% RSLogix 500 project VA116HF7_OPRAVOVANY_4_2017_02_12.rss, saved by version 8.40.00.08 %
PROJECT "VA116"    % processor: SLC 500, 1747-L532; 601760_CO2 %

PROGRAM FILES
  LAD 2 "601760_CO2"  92 rungs
  LAD 3   24 rungs
  LAD 4   108 rungs
  LAD 5   16 rungs
  LAD 6   98 rungs
  LAD 7   26 rungs
  LAD 8   13 rungs
  LAD 9   15 rungs
  LAD 10   50 rungs
  LAD 11   95 rungs
  LAD 12   18 rungs
  LAD 13   34 rungs
  LAD 14   6 rungs
  LAD 15   28 rungs
  LAD 16   84 rungs
  LAD 17   22 rungs
  LAD 18   23 rungs
  LAD 19   37 rungs
  LAD 20   5 rungs
  LAD 21   19 rungs
  LAD 22   29 rungs
  LAD 23   17 rungs
  LAD 24   32 rungs
  LAD 25   8 rungs
  LAD 26   57 rungs
  LAD 27   4 rungs
  LAD 28   3 rungs
  LAD 29   4 rungs
  LAD 30   12 rungs
  LAD 31   12 rungs
  LAD 32   22 rungs
  LAD 33   10 rungs
  LAD 34   16 rungs
  LAD 35   14 rungs

DATA FILES
  O0 OUTPUT  4 elements
  I1 INPUT  8 elements
  S2 STATUS  83 elements
  B3 BINARY  1 elements
  T4 TIMER  61 elements
  C5 COUNTER  6 elements
  R6 CONTROL  1 elements
  N7 INTEGER  110 elements
  N10   256 elements
  N11   256 elements

LADDER 2 "601760_CO2"
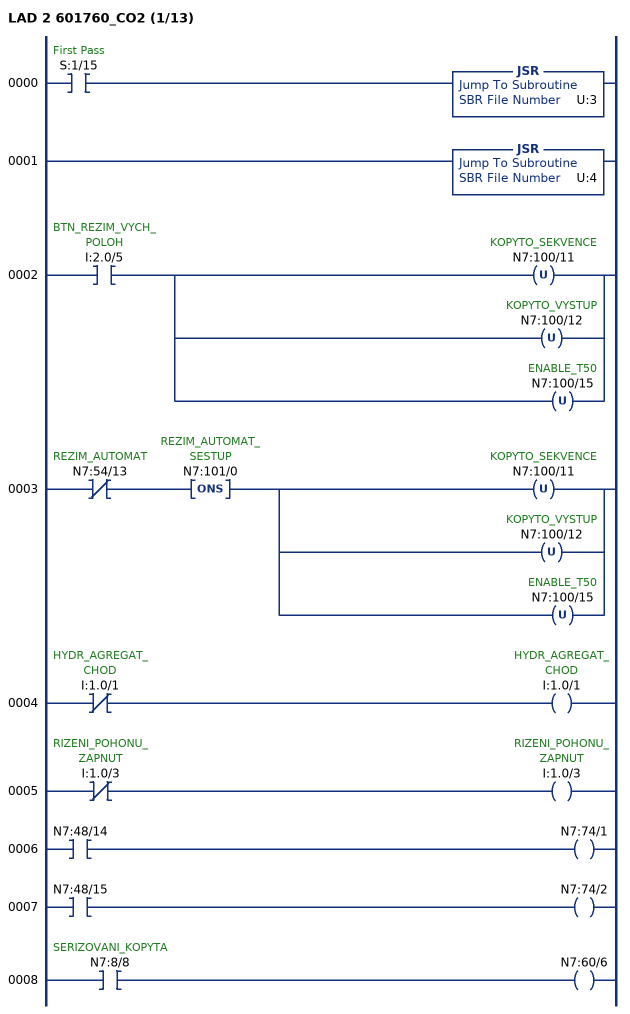
% Rung: 0 %
SOR XIC S:1/15 JSR U:3 EOR
%   S:1/15  "First Pass" %
% Rung: 1 %
SOR JSR U:4 EOR
% Rung: 2 %
SOR XIC I:2.0/5 BST OTU N7:100/11 NXB OTU N7:100/12 NXB OTU N7:100/15 BND EOR
%   I:2.0/5  BTN_REZIM_VYCH_POLOH %
%   N7:100/11  KOPYTO_SEKVENCE %
%   N7:100/12  KOPYTO_VYSTUP %
%   N7:100/15  ENABLE_T50 %
% Rung: 3 %
SOR XIO N7:54/13 OSR N7:101/0 BST OTU N7:100/11 NXB OTU N7:100/12 NXB OTU N7:100/15 BND EOR
%   N7:54/13  REZIM_AUTOMAT %
%   N7:101/0  REZIM_AUTOMAT_SESTUP %
%   N7:100/11  KOPYTO_SEKVENCE %
%   N7:100/12  KOPYTO_VYSTUP %
%   N7:100/15  ENABLE_T50 %
% Rung: 4 %
SOR XIO I:1.0/1 OTE I:1.0/1 EOR
%   I:1.0/1  HYDR_AGREGAT_CHOD %
% Rung: 5 %
SOR XIO I:1.0/3 OTE I:1.0/3 EOR
%   I:1.0/3  RIZENI_POHONU_ZAPNUT %
% Rung: 6 %
SOR XIC N7:48/14 OTE N7:74/1 EOR
% Rung: 7 %
SOR XIC N7:48/15 OTE N7:74/2 EOR
% Rung: 8 %
SOR XIC N7:8/8 OTE N7:60/6 EOR
%   N7:8/8  SERIZOVANI_KOPYTA %

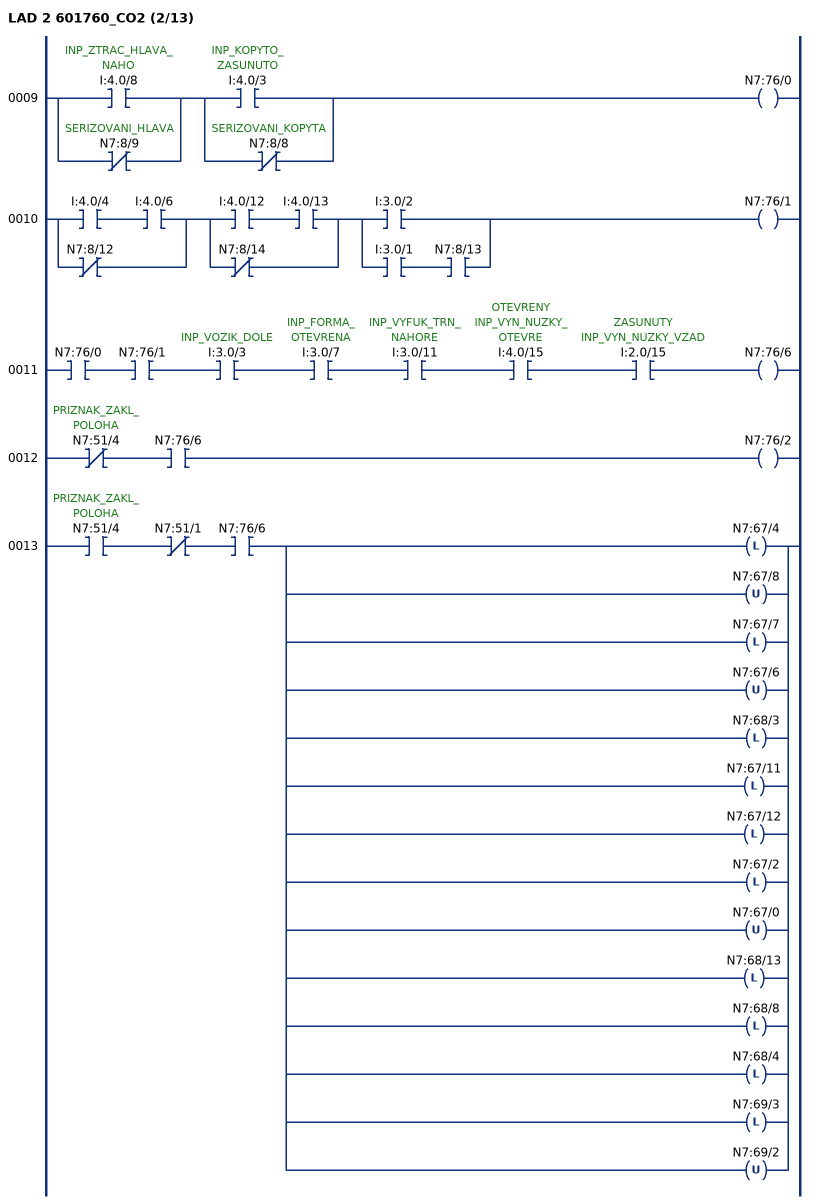
% Rung: 9 %
SOR BST XIC I:4.0/8 NXB XIO N7:8/9 BND BST XIC I:4.0/3 NXB XIO N7:8/8 BND OTE N7:76/0 EOR
%   I:4.0/8  INP_ZTRAC_HLAVA_NAHO %
%   N7:8/9  SERIZOVANI_HLAVA %
%   I:4.0/3  INP_KOPYTO_ZASUNUTO %
%   N7:8/8  SERIZOVANI_KOPYTA %
% Rung: 10 %
SOR BST XIC I:4.0/4 XIC I:4.0/6 NXB XIO N7:8/12 BND BST XIC I:4.0/12 XIC I:4.0/13 NXB XIO N7:8/14 BND BST XIC I:3.0/2 NXB XIC I:3.0/1 XIC N7:8/13 BND OTE N7:76/1 EOR
% Rung: 11 %
SOR XIC N7:76/0 XIC N7:76/1 XIC I:3.0/3 XIC I:3.0/7 XIC I:3.0/11 XIC I:4.0/15 XIC I:2.0/15 OTE N7:76/6 EOR
%   I:3.0/3  INP_VOZIK_DOLE %
%   I:3.0/7  INP_FORMA_OTEVRENA %
%   I:3.0/11  INP_VYFUK_TRN_NAHORE %
%   I:4.0/15  INP_VYN_NUZKY_OTEVRE  "OTEVRENY" %
%   I:2.0/15  INP_VYN_NUZKY_VZAD  "ZASUNUTY" %
% Rung: 12 %
SOR XIO N7:51/4 XIC N7:76/6 OTE N7:76/2 EOR
%   N7:51/4  PRIZNAK_ZAKL_POLOHA %
% Rung: 13 %
SOR XIC N7:51/4 XIO N7:51/1 XIC N7:76/6 BST OTL N7:67/4 NXB OTU N7:67/8 NXB BST OTL N7:67/7 NXB OTU N7:67/6 BND NXB OTL N7:68/3 NXB OTL N7:67/11 NXB OTL N7:67/12 NXB OTL N7:67/2 NXB OTU N7:67/0 NXB OTL N7:68/13 NXB OTL N7:68/8 NXB BST OTL N7:68/4 NXB BST OTL N7:69/3 NXB OTU N7:69/2 BND BND BND EOR
%   N7:51/4  PRIZNAK_ZAKL_POLOHA %

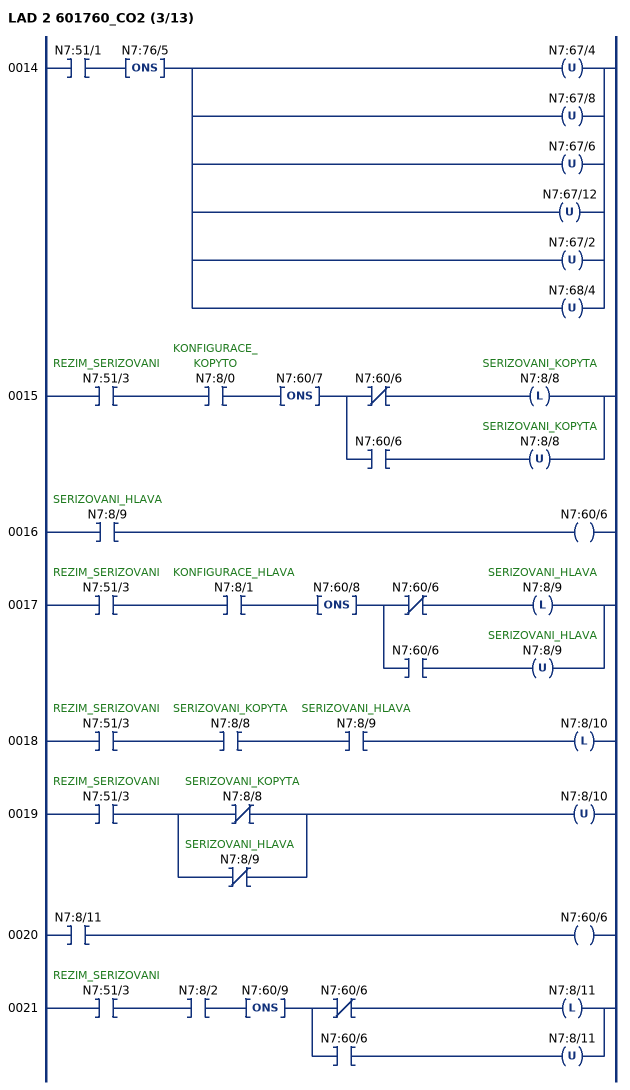
% Rung: 14 %
SOR XIC N7:51/1 OSR N7:76/5 BST OTU N7:67/4 NXB OTU N7:67/8 NXB OTU N7:67/6 NXB OTU N7:67/12 NXB OTU N7:67/2 NXB OTU N7:68/4 BND EOR
% Rung: 15 %
SOR XIC N7:51/3 XIC N7:8/0 OSR N7:60/7 BST XIO N7:60/6 OTL N7:8/8 NXB XIC N7:60/6 OTU N7:8/8 BND EOR
%   N7:51/3  REZIM_SERIZOVANI %
%   N7:8/0  KONFIGURACE_KOPYTO %
%   N7:8/8  SERIZOVANI_KOPYTA %
% Rung: 16 %
SOR XIC N7:8/9 OTE N7:60/6 EOR
%   N7:8/9  SERIZOVANI_HLAVA %
% Rung: 17 %
SOR XIC N7:51/3 XIC N7:8/1 OSR N7:60/8 BST XIO N7:60/6 OTL N7:8/9 NXB XIC N7:60/6 OTU N7:8/9 BND EOR
%   N7:51/3  REZIM_SERIZOVANI %
%   N7:8/1  KONFIGURACE_HLAVA %
%   N7:8/9  SERIZOVANI_HLAVA %
% Rung: 18 %
SOR XIC N7:51/3 XIC N7:8/8 XIC N7:8/9 OTL N7:8/10 EOR
%   N7:51/3  REZIM_SERIZOVANI %
%   N7:8/8  SERIZOVANI_KOPYTA %
%   N7:8/9  SERIZOVANI_HLAVA %
% Rung: 19 %
SOR XIC N7:51/3 BST XIO N7:8/8 NXB XIO N7:8/9 BND OTU N7:8/10 EOR
%   N7:51/3  REZIM_SERIZOVANI %
%   N7:8/8  SERIZOVANI_KOPYTA %
%   N7:8/9  SERIZOVANI_HLAVA %
% Rung: 20 %
SOR XIC N7:8/11 OTE N7:60/6 EOR
% Rung: 21 %
SOR XIC N7:51/3 XIC N7:8/2 OSR N7:60/9 BST XIO N7:60/6 OTL N7:8/11 NXB XIC N7:60/6 OTU N7:8/11 BND EOR
%   N7:51/3  REZIM_SERIZOVANI %

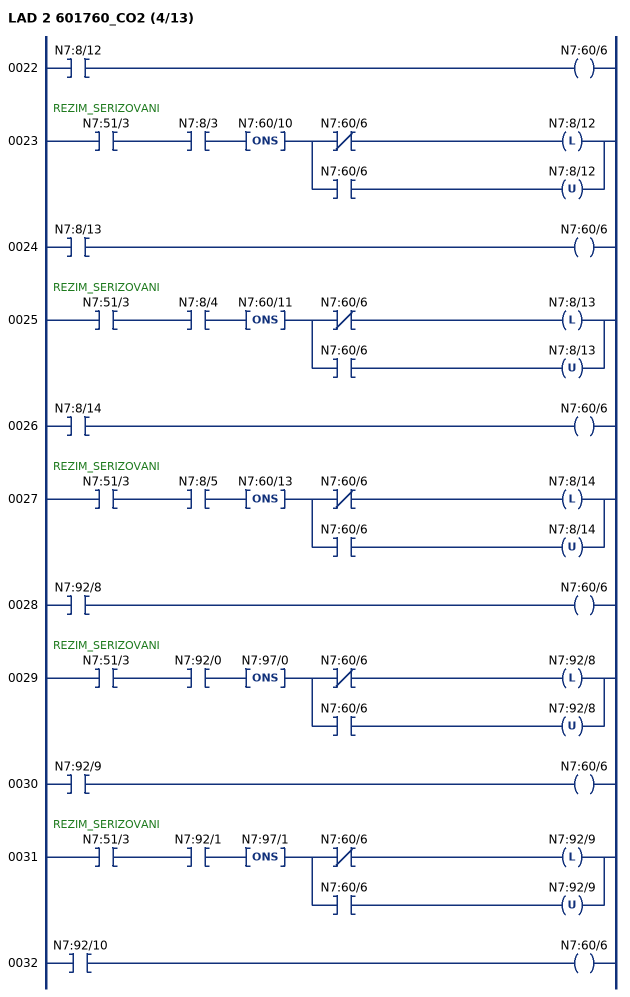
% Rung: 22 %
SOR XIC N7:8/12 OTE N7:60/6 EOR
% Rung: 23 %
SOR XIC N7:51/3 XIC N7:8/3 OSR N7:60/10 BST XIO N7:60/6 OTL N7:8/12 NXB XIC N7:60/6 OTU N7:8/12 BND EOR
%   N7:51/3  REZIM_SERIZOVANI %
% Rung: 24 %
SOR XIC N7:8/13 OTE N7:60/6 EOR
% Rung: 25 %
SOR XIC N7:51/3 XIC N7:8/4 OSR N7:60/11 BST XIO N7:60/6 OTL N7:8/13 NXB XIC N7:60/6 OTU N7:8/13 BND EOR
%   N7:51/3  REZIM_SERIZOVANI %
% Rung: 26 %
SOR XIC N7:8/14 OTE N7:60/6 EOR
% Rung: 27 %
SOR XIC N7:51/3 XIC N7:8/5 OSR N7:60/13 BST XIO N7:60/6 OTL N7:8/14 NXB XIC N7:60/6 OTU N7:8/14 BND EOR
%   N7:51/3  REZIM_SERIZOVANI %
% Rung: 28 %
SOR XIC N7:92/8 OTE N7:60/6 EOR
% Rung: 29 %
SOR XIC N7:51/3 XIC N7:92/0 OSR N7:97/0 BST XIO N7:60/6 OTL N7:92/8 NXB XIC N7:60/6 OTU N7:92/8 BND EOR
%   N7:51/3  REZIM_SERIZOVANI %
% Rung: 30 %
SOR XIC N7:92/9 OTE N7:60/6 EOR
% Rung: 31 %
SOR XIC N7:51/3 XIC N7:92/1 OSR N7:97/1 BST XIO N7:60/6 OTL N7:92/9 NXB XIC N7:60/6 OTU N7:92/9 BND EOR
%   N7:51/3  REZIM_SERIZOVANI %
% Rung: 32 %
SOR XIC N7:92/10 OTE N7:60/6 EOR

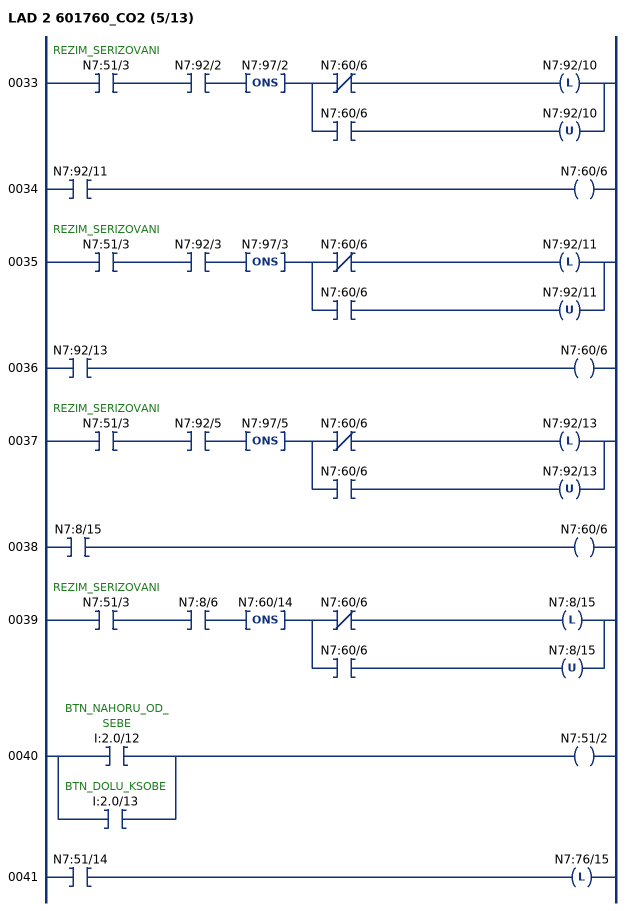
% Rung: 33 %
SOR XIC N7:51/3 XIC N7:92/2 OSR N7:97/2 BST XIO N7:60/6 OTL N7:92/10 NXB XIC N7:60/6 OTU N7:92/10 BND EOR
%   N7:51/3  REZIM_SERIZOVANI %
% Rung: 34 %
SOR XIC N7:92/11 OTE N7:60/6 EOR
% Rung: 35 %
SOR XIC N7:51/3 XIC N7:92/3 OSR N7:97/3 BST XIO N7:60/6 OTL N7:92/11 NXB XIC N7:60/6 OTU N7:92/11 BND EOR
%   N7:51/3  REZIM_SERIZOVANI %
% Rung: 36 %
SOR XIC N7:92/13 OTE N7:60/6 EOR
% Rung: 37 %
SOR XIC N7:51/3 XIC N7:92/5 OSR N7:97/5 BST XIO N7:60/6 OTL N7:92/13 NXB XIC N7:60/6 OTU N7:92/13 BND EOR
%   N7:51/3  REZIM_SERIZOVANI %
% Rung: 38 %
SOR XIC N7:8/15 OTE N7:60/6 EOR
% Rung: 39 %
SOR XIC N7:51/3 XIC N7:8/6 OSR N7:60/14 BST XIO N7:60/6 OTL N7:8/15 NXB XIC N7:60/6 OTU N7:8/15 BND EOR
%   N7:51/3  REZIM_SERIZOVANI %
% Rung: 40 %
SOR BST XIC I:2.0/12 NXB XIC I:2.0/13 BND OTE N7:51/2 EOR
%   I:2.0/12  BTN_NAHORU_OD_SEBE %
%   I:2.0/13  BTN_DOLU_KSOBE %
% Rung: 41 %
SOR XIC N7:51/14 OTL N7:76/15 EOR

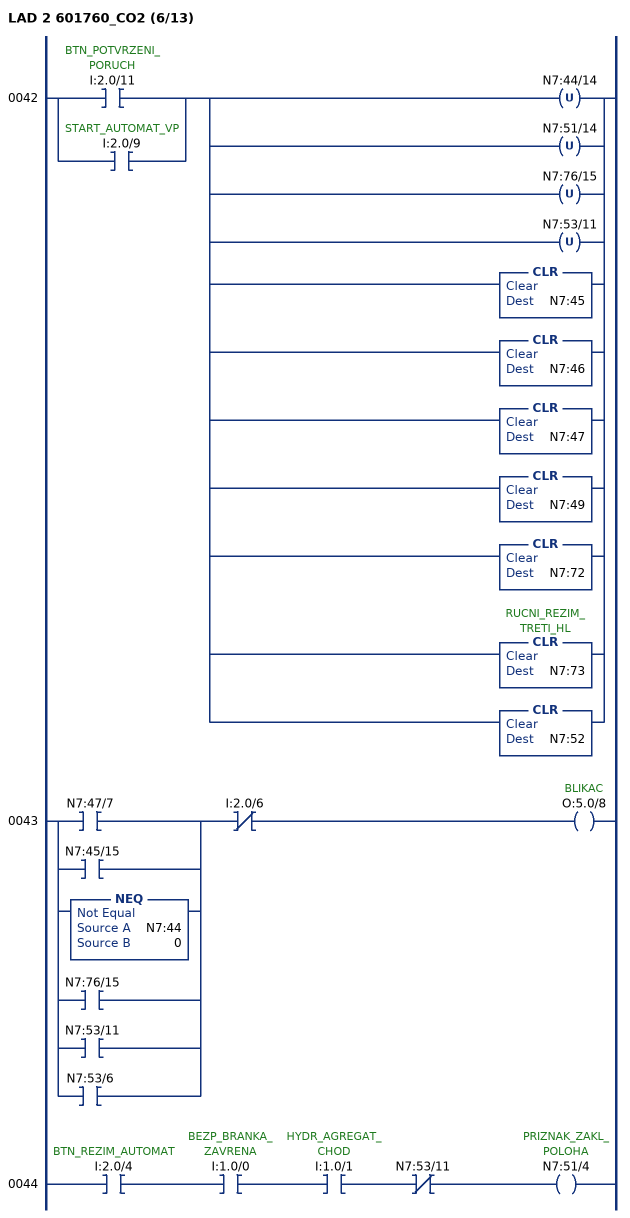
% Rung: 42 %
SOR BST XIC I:2.0/11 NXB XIC I:2.0/9 BND BST OTU N7:44/14 NXB OTU N7:51/14 NXB OTU N7:76/15 NXB OTU N7:53/11 NXB CLR N7:45 NXB CLR N7:46 NXB CLR N7:47 NXB CLR N7:49 NXB CLR N7:72 NXB CLR N7:73 NXB CLR N7:52 BND EOR
%   I:2.0/11  BTN_POTVRZENI_PORUCH %
%   I:2.0/9  START_AUTOMAT_VP %
%   N7:73  RUCNI_REZIM_TRETI_HL %
% Rung: 43 %
SOR BST XIC N7:47/7 NXB XIC N7:45/15 NXB NEQ N7:44 0 NXB XIC N7:76/15 NXB XIC N7:53/11 NXB XIC N7:53/6 BND XIO I:2.0/6 OTE O:5.0/8 EOR
%   O:5.0/8  BLIKAC %
% Rung: 44 %
SOR XIC I:2.0/4 XIC I:1.0/0 XIC I:1.0/1 XIO N7:53/11 OTE N7:51/4 EOR
%   I:2.0/4  BTN_REZIM_AUTOMAT %
%   I:1.0/0  BEZP_BRANKA_ZAVRENA %
%   I:1.0/1  HYDR_AGREGAT_CHOD %
%   N7:51/4  PRIZNAK_ZAKL_POLOHA %

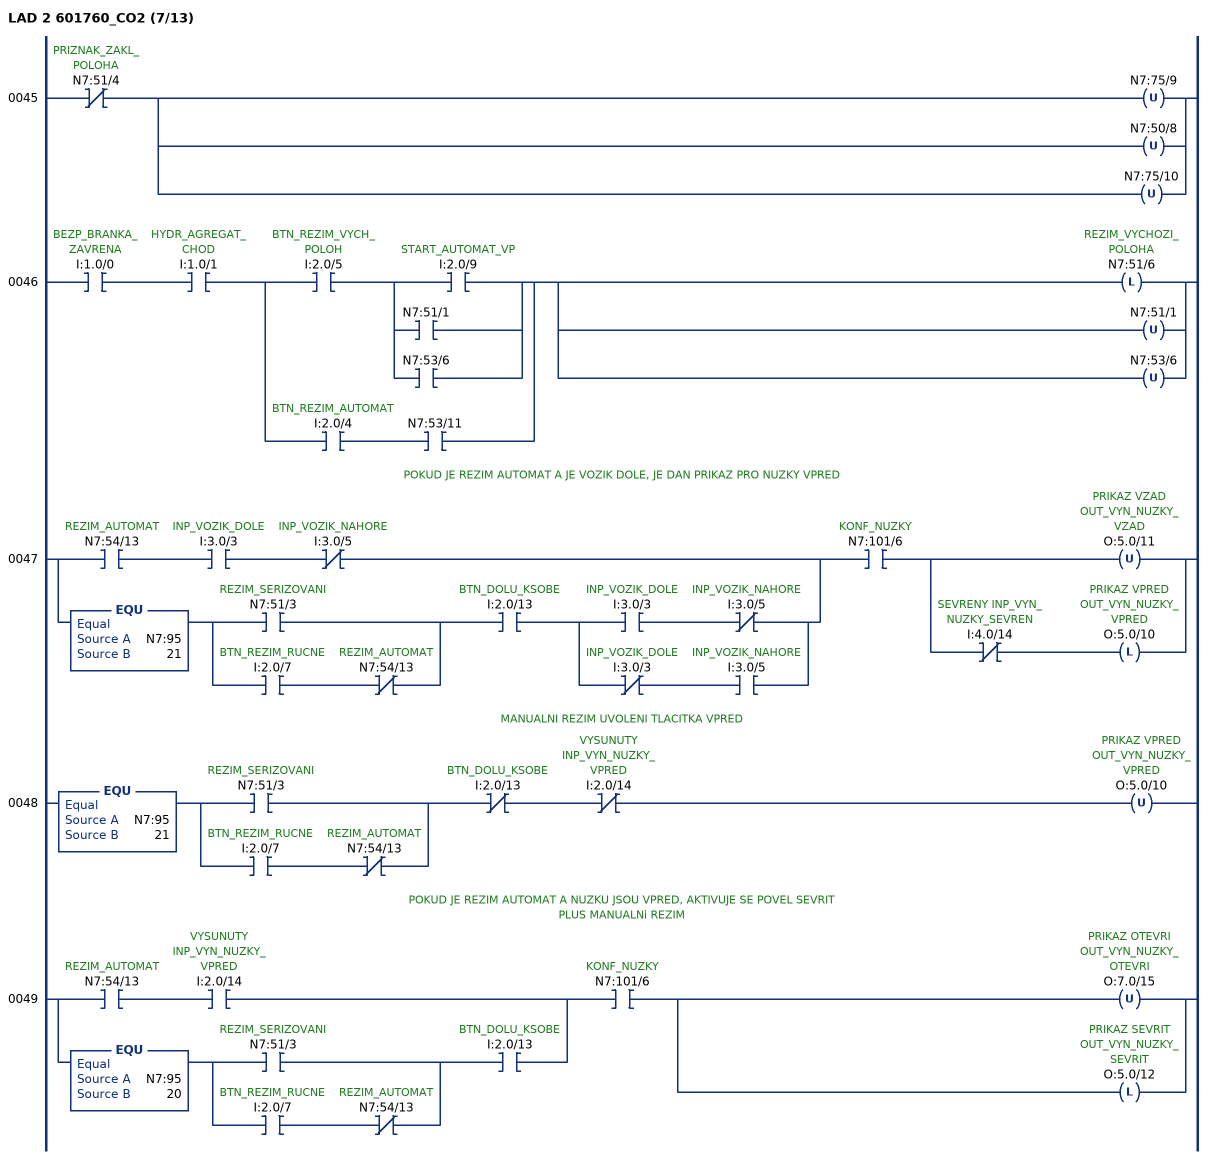
% Rung: 45 %
SOR XIO N7:51/4 BST OTU N7:75/9 NXB OTU N7:50/8 NXB OTU N7:75/10 BND EOR
%   N7:51/4  PRIZNAK_ZAKL_POLOHA %
% Rung: 46 %
SOR XIC I:1.0/0 XIC I:1.0/1 BST XIC I:2.0/5 BST XIC I:2.0/9 NXB XIC N7:51/1 NXB XIC N7:53/6 BND NXB XIC I:2.0/4 XIC N7:53/11 BND BST OTL N7:51/6 NXB OTU N7:51/1 NXB OTU N7:53/6 BND EOR
%   I:1.0/0  BEZP_BRANKA_ZAVRENA %
%   I:1.0/1  HYDR_AGREGAT_CHOD %
%   I:2.0/5  BTN_REZIM_VYCH_POLOH %
%   I:2.0/9  START_AUTOMAT_VP %
%   I:2.0/4  BTN_REZIM_AUTOMAT %
%   N7:51/6  REZIM_VYCHOZI_POLOHA %
% Rung: 47 %
% POKUD JE REZIM AUTOMAT A JE VOZIK DOLE, JE DAN PRIKAZ PRO NUZKY VPRED %
SOR BST XIC N7:54/13 XIC I:3.0/3 XIO I:3.0/5 NXB EQU N7:95 21 BST XIC N7:51/3 NXB XIC I:2.0/7 XIO N7:54/13 BND XIC I:2.0/13 BST XIC I:3.0/3 XIO I:3.0/5 NXB XIO I:3.0/3 XIC I:3.0/5 BND BND XIC N7:101/6 BST OTU O:5.0/11 NXB XIO I:4.0/14 OTL O:5.0/10 BND EOR
%   N7:54/13  REZIM_AUTOMAT %
%   I:3.0/3  INP_VOZIK_DOLE %
%   I:3.0/5  INP_VOZIK_NAHORE %
%   N7:51/3  REZIM_SERIZOVANI %
%   I:2.0/7  BTN_REZIM_RUCNE %
%   I:2.0/13  BTN_DOLU_KSOBE %
%   N7:101/6  KONF_NUZKY %
%   O:5.0/11  OUT_VYN_NUZKY_VZAD  "PRIKAZ VZAD" %
%   I:4.0/14  INP_VYN_NUZKY_SEVREN  "SEVRENY" %
%   O:5.0/10  OUT_VYN_NUZKY_VPRED  "PRIKAZ VPRED" %
% Rung: 48 %
% MANUALNI REZIM UVOLENI TLACITKA VPRED %
SOR EQU N7:95 21 BST XIC N7:51/3 NXB XIC I:2.0/7 XIO N7:54/13 BND XIO I:2.0/13 XIO I:2.0/14 OTU O:5.0/10 EOR
%   N7:51/3  REZIM_SERIZOVANI %
%   I:2.0/7  BTN_REZIM_RUCNE %
%   N7:54/13  REZIM_AUTOMAT %
%   I:2.0/13  BTN_DOLU_KSOBE %
%   I:2.0/14  INP_VYN_NUZKY_VPRED  "VYSUNUTY" %
%   O:5.0/10  OUT_VYN_NUZKY_VPRED  "PRIKAZ VPRED" %
% Rung: 49 %
% POKUD JE REZIM AUTOMAT A NUZKU JSOU VPRED, AKTIVUJE SE POVEL SEVRIT
% PLUS MANUALNi REZIM %
SOR BST XIC N7:54/13 XIC I:2.0/14 NXB EQU N7:95 20 BST XIC N7:51/3 NXB XIC I:2.0/7 XIO N7:54/13 BND XIC I:2.0/13 BND XIC N7:101/6 BST OTU O:7.0/15 NXB OTL O:5.0/12 BND EOR
%   N7:54/13  REZIM_AUTOMAT %
%   I:2.0/14  INP_VYN_NUZKY_VPRED  "VYSUNUTY" %
%   N7:51/3  REZIM_SERIZOVANI %
%   I:2.0/7  BTN_REZIM_RUCNE %
%   I:2.0/13  BTN_DOLU_KSOBE %
%   N7:101/6  KONF_NUZKY %
%   O:7.0/15  OUT_VYN_NUZKY_OTEVRI  "PRIKAZ OTEVRI" %
%   O:5.0/12  OUT_VYN_NUZKY_SEVRIT  "PRIKAZ SEVRIT" %

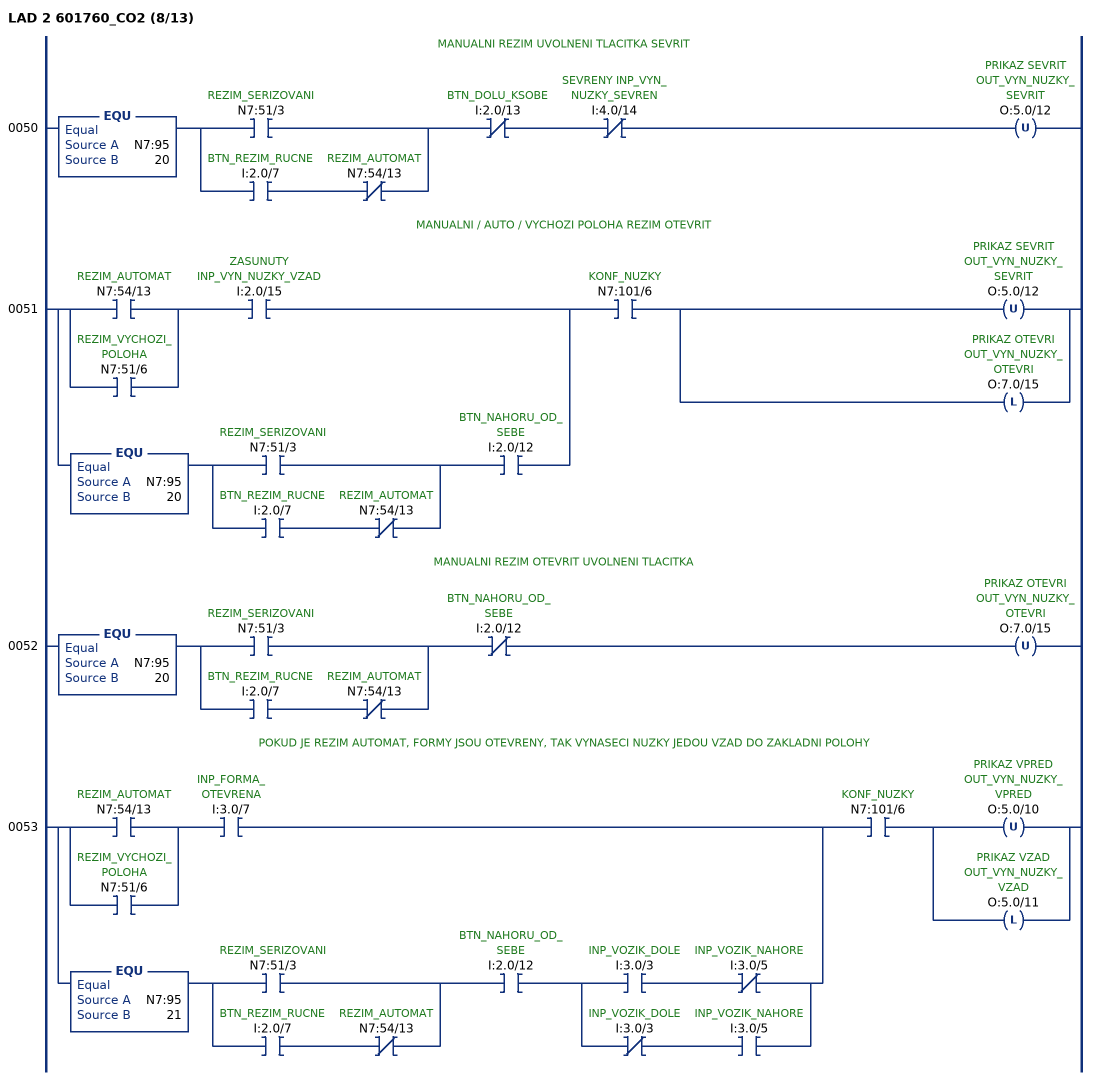
% Rung: 50 %
% MANUALNI REZIM UVOLNENI TLACITKA SEVRIT %
SOR EQU N7:95 20 BST XIC N7:51/3 NXB XIC I:2.0/7 XIO N7:54/13 BND XIO I:2.0/13 XIO I:4.0/14 OTU O:5.0/12 EOR
%   N7:51/3  REZIM_SERIZOVANI %
%   I:2.0/7  BTN_REZIM_RUCNE %
%   N7:54/13  REZIM_AUTOMAT %
%   I:2.0/13  BTN_DOLU_KSOBE %
%   I:4.0/14  INP_VYN_NUZKY_SEVREN  "SEVRENY" %
%   O:5.0/12  OUT_VYN_NUZKY_SEVRIT  "PRIKAZ SEVRIT" %
% Rung: 51 %
% MANUALNI / AUTO / VYCHOZI POLOHA REZIM OTEVRIT %
SOR BST BST XIC N7:54/13 NXB XIC N7:51/6 BND XIC I:2.0/15 NXB EQU N7:95 20 BST XIC N7:51/3 NXB XIC I:2.0/7 XIO N7:54/13 BND XIC I:2.0/12 BND XIC N7:101/6 BST OTU O:5.0/12 NXB OTL O:7.0/15 BND EOR
%   N7:54/13  REZIM_AUTOMAT %
%   N7:51/6  REZIM_VYCHOZI_POLOHA %
%   I:2.0/15  INP_VYN_NUZKY_VZAD  "ZASUNUTY" %
%   N7:51/3  REZIM_SERIZOVANI %
%   I:2.0/7  BTN_REZIM_RUCNE %
%   I:2.0/12  BTN_NAHORU_OD_SEBE %
%   N7:101/6  KONF_NUZKY %
%   O:5.0/12  OUT_VYN_NUZKY_SEVRIT  "PRIKAZ SEVRIT" %
%   O:7.0/15  OUT_VYN_NUZKY_OTEVRI  "PRIKAZ OTEVRI" %
% Rung: 52 %
% MANUALNI REZIM OTEVRIT UVOLNENI TLACITKA %
SOR EQU N7:95 20 BST XIC N7:51/3 NXB XIC I:2.0/7 XIO N7:54/13 BND XIO I:2.0/12 OTU O:7.0/15 EOR
%   N7:51/3  REZIM_SERIZOVANI %
%   I:2.0/7  BTN_REZIM_RUCNE %
%   N7:54/13  REZIM_AUTOMAT %
%   I:2.0/12  BTN_NAHORU_OD_SEBE %
%   O:7.0/15  OUT_VYN_NUZKY_OTEVRI  "PRIKAZ OTEVRI" %
% Rung: 53 %
% POKUD JE REZIM AUTOMAT, FORMY JSOU OTEVRENY, TAK VYNASECI NUZKY JEDOU VZAD DO ZAKLADNI POLOHY %
SOR BST BST XIC N7:54/13 NXB XIC N7:51/6 BND XIC I:3.0/7 NXB EQU N7:95 21 BST XIC N7:51/3 NXB XIC I:2.0/7 XIO N7:54/13 BND XIC I:2.0/12 BST XIC I:3.0/3 XIO I:3.0/5 NXB XIO I:3.0/3 XIC I:3.0/5 BND BND XIC N7:101/6 BST OTU O:5.0/10 NXB OTL O:5.0/11 BND EOR
%   N7:54/13  REZIM_AUTOMAT %
%   N7:51/6  REZIM_VYCHOZI_POLOHA %
%   I:3.0/7  INP_FORMA_OTEVRENA %
%   N7:51/3  REZIM_SERIZOVANI %
%   I:2.0/7  BTN_REZIM_RUCNE %
%   I:2.0/12  BTN_NAHORU_OD_SEBE %
%   I:3.0/3  INP_VOZIK_DOLE %
%   I:3.0/5  INP_VOZIK_NAHORE %
%   N7:101/6  KONF_NUZKY %
%   O:5.0/10  OUT_VYN_NUZKY_VPRED  "PRIKAZ VPRED" %
%   O:5.0/11  OUT_VYN_NUZKY_VZAD  "PRIKAZ VZAD" %

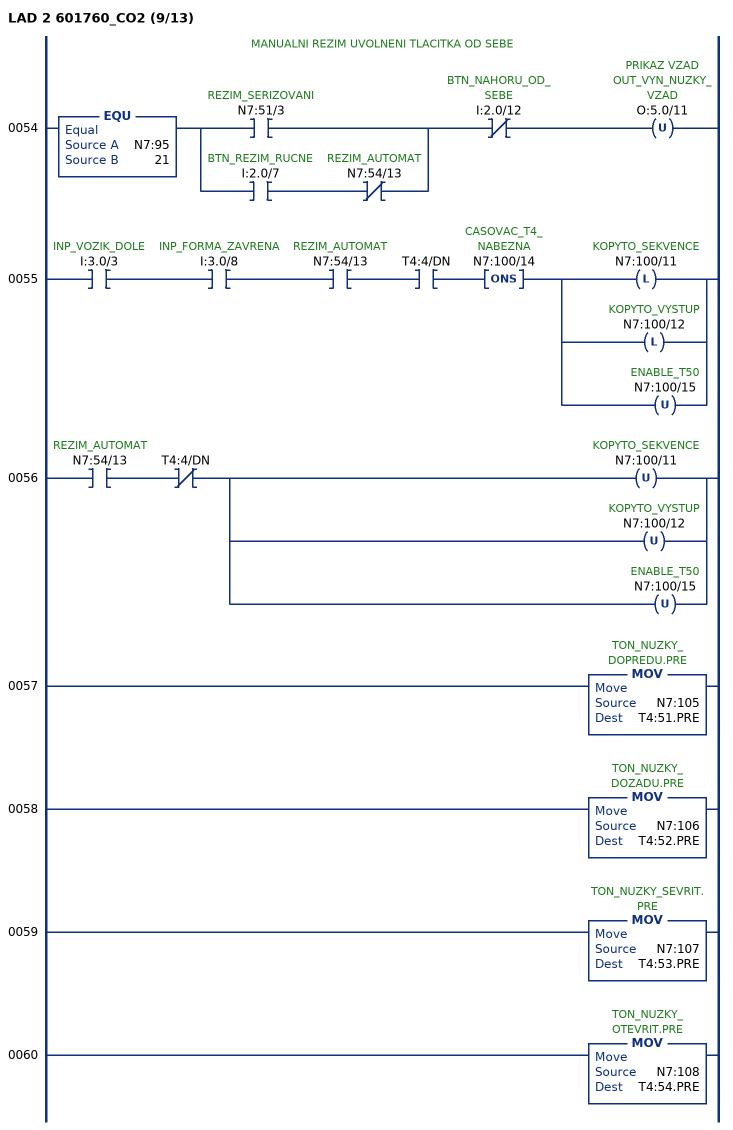
% Rung: 54 %
% MANUALNI REZIM UVOLNENI TLACITKA OD SEBE %
SOR EQU N7:95 21 BST XIC N7:51/3 NXB XIC I:2.0/7 XIO N7:54/13 BND XIO I:2.0/12 OTU O:5.0/11 EOR
%   N7:51/3  REZIM_SERIZOVANI %
%   I:2.0/7  BTN_REZIM_RUCNE %
%   N7:54/13  REZIM_AUTOMAT %
%   I:2.0/12  BTN_NAHORU_OD_SEBE %
%   O:5.0/11  OUT_VYN_NUZKY_VZAD  "PRIKAZ VZAD" %
% Rung: 55 %
SOR XIC I:3.0/3 XIC I:3.0/8 XIC N7:54/13 XIC T4:4/DN OSR N7:100/14 BST OTL N7:100/11 NXB OTL N7:100/12 NXB OTU N7:100/15 BND EOR
%   I:3.0/3  INP_VOZIK_DOLE %
%   I:3.0/8  INP_FORMA_ZAVRENA %
%   N7:54/13  REZIM_AUTOMAT %
%   N7:100/14  CASOVAC_T4_NABEZNA %
%   N7:100/11  KOPYTO_SEKVENCE %
%   N7:100/12  KOPYTO_VYSTUP %
%   N7:100/15  ENABLE_T50 %
% Rung: 56 %
SOR XIC N7:54/13 XIO T4:4/DN BST OTU N7:100/11 NXB OTU N7:100/12 NXB OTU N7:100/15 BND EOR
%   N7:54/13  REZIM_AUTOMAT %
%   N7:100/11  KOPYTO_SEKVENCE %
%   N7:100/12  KOPYTO_VYSTUP %
%   N7:100/15  ENABLE_T50 %
% Rung: 57 %
SOR MOV N7:105 T4:51.PRE EOR
%   N7:105  CASOVAC_T51_PRESET %
%   T4:51  TON_NUZKY_DOPREDU %
% Rung: 58 %
SOR MOV N7:106 T4:52.PRE EOR
%   N7:106  CASOVAC_T52_PRESET %
%   T4:52  TON_NUZKY_DOZADU %
% Rung: 59 %
SOR MOV N7:107 T4:53.PRE EOR
%   N7:107  CASOVAC_T53_PRESET %
%   T4:53  TON_NUZKY_SEVRIT %
% Rung: 60 %
SOR MOV N7:108 T4:54.PRE EOR
%   N7:108  CASOVAC_T54_PRESET %
%   T4:54  TON_NUZKY_OTEVRIT %

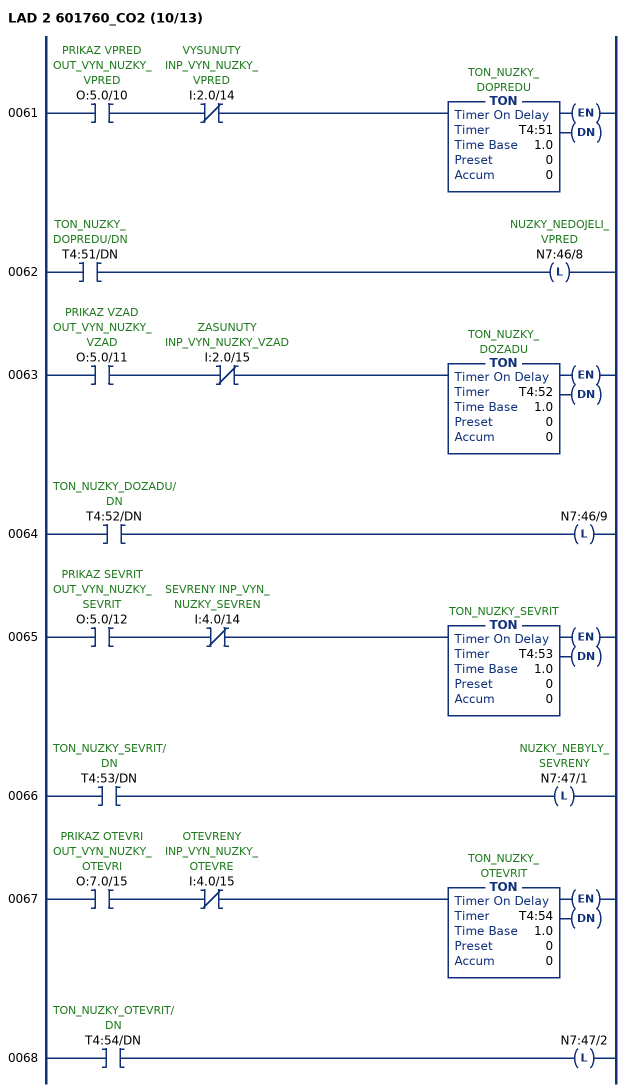
% Rung: 61 %
SOR XIC O:5.0/10 XIO I:2.0/14 TON T4:51 1.0 0 0 EOR
%   O:5.0/10  OUT_VYN_NUZKY_VPRED  "PRIKAZ VPRED" %
%   I:2.0/14  INP_VYN_NUZKY_VPRED  "VYSUNUTY" %
%   T4:51  TON_NUZKY_DOPREDU %
% Rung: 62 %
SOR XIC T4:51/DN OTL N7:46/8 EOR
%   T4:51  TON_NUZKY_DOPREDU %
%   N7:46/8  NUZKY_NEDOJELI_VPRED %
% Rung: 63 %
SOR XIC O:5.0/11 XIO I:2.0/15 TON T4:52 1.0 0 0 EOR
%   O:5.0/11  OUT_VYN_NUZKY_VZAD  "PRIKAZ VZAD" %
%   I:2.0/15  INP_VYN_NUZKY_VZAD  "ZASUNUTY" %
%   T4:52  TON_NUZKY_DOZADU %
% Rung: 64 %
SOR XIC T4:52/DN OTL N7:46/9 EOR
%   T4:52  TON_NUZKY_DOZADU %
% Rung: 65 %
SOR XIC O:5.0/12 XIO I:4.0/14 TON T4:53 1.0 0 0 EOR
%   O:5.0/12  OUT_VYN_NUZKY_SEVRIT  "PRIKAZ SEVRIT" %
%   I:4.0/14  INP_VYN_NUZKY_SEVREN  "SEVRENY" %
%   T4:53  TON_NUZKY_SEVRIT %
% Rung: 66 %
SOR XIC T4:53/DN OTL N7:47/1 EOR
%   T4:53  TON_NUZKY_SEVRIT %
%   N7:47/1  NUZKY_NEBYLY_SEVRENY %
% Rung: 67 %
SOR XIC O:7.0/15 XIO I:4.0/15 TON T4:54 1.0 0 0 EOR
%   O:7.0/15  OUT_VYN_NUZKY_OTEVRI  "PRIKAZ OTEVRI" %
%   I:4.0/15  INP_VYN_NUZKY_OTEVRE  "OTEVRENY" %
%   T4:54  TON_NUZKY_OTEVRIT %
% Rung: 68 %
SOR XIC T4:54/DN OTL N7:47/2 EOR
%   T4:54  TON_NUZKY_OTEVRIT %

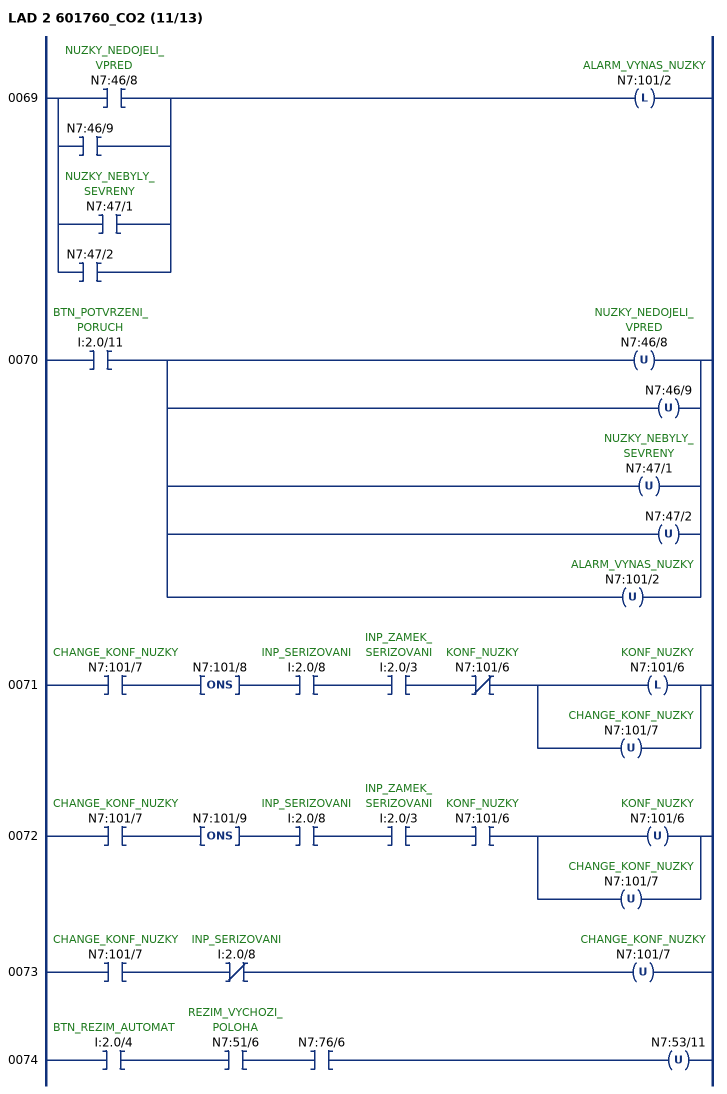
% Rung: 69 %
SOR BST XIC N7:46/8 NXB XIC N7:46/9 NXB XIC N7:47/1 NXB XIC N7:47/2 BND OTL N7:101/2 EOR
%   N7:46/8  NUZKY_NEDOJELI_VPRED %
%   N7:47/1  NUZKY_NEBYLY_SEVRENY %
%   N7:101/2  ALARM_VYNAS_NUZKY %
% Rung: 70 %
SOR XIC I:2.0/11 BST OTU N7:46/8 NXB OTU N7:46/9 NXB OTU N7:47/1 NXB OTU N7:47/2 NXB OTU N7:101/2 BND EOR
%   I:2.0/11  BTN_POTVRZENI_PORUCH %
%   N7:46/8  NUZKY_NEDOJELI_VPRED %
%   N7:47/1  NUZKY_NEBYLY_SEVRENY %
%   N7:101/2  ALARM_VYNAS_NUZKY %
% Rung: 71 %
SOR XIC N7:101/7 OSR N7:101/8 XIC I:2.0/8 XIC I:2.0/3 XIO N7:101/6 BST OTL N7:101/6 NXB OTU N7:101/7 BND EOR
%   N7:101/7  CHANGE_KONF_NUZKY %
%   I:2.0/8  INP_SERIZOVANI %
%   I:2.0/3  INP_ZAMEK_SERIZOVANI %
%   N7:101/6  KONF_NUZKY %
% Rung: 72 %
SOR XIC N7:101/7 OSR N7:101/9 XIC I:2.0/8 XIC I:2.0/3 XIC N7:101/6 BST OTU N7:101/6 NXB OTU N7:101/7 BND EOR
%   N7:101/7  CHANGE_KONF_NUZKY %
%   I:2.0/8  INP_SERIZOVANI %
%   I:2.0/3  INP_ZAMEK_SERIZOVANI %
%   N7:101/6  KONF_NUZKY %
% Rung: 73 %
SOR XIC N7:101/7 XIO I:2.0/8 OTU N7:101/7 EOR
%   N7:101/7  CHANGE_KONF_NUZKY %
%   I:2.0/8  INP_SERIZOVANI %
% Rung: 74 %
SOR XIC I:2.0/4 XIC N7:51/6 XIC N7:76/6 OTU N7:53/11 EOR
%   I:2.0/4  BTN_REZIM_AUTOMAT %
%   N7:51/6  REZIM_VYCHOZI_POLOHA %

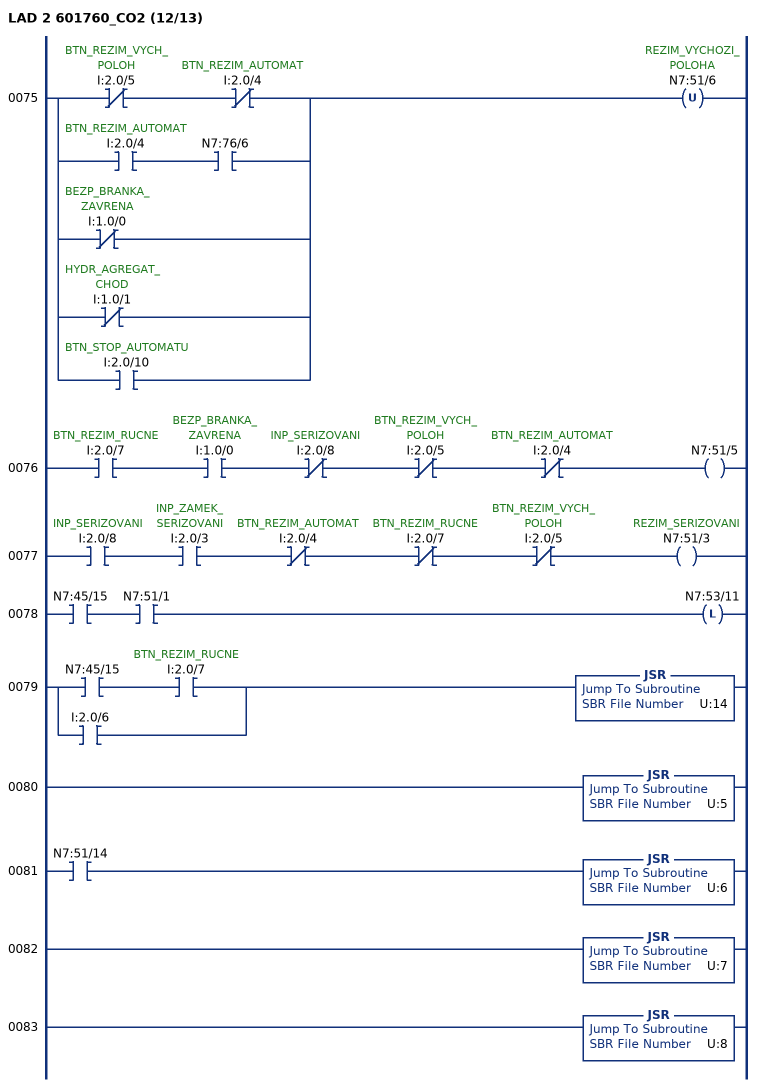
% Rung: 75 %
SOR BST XIO I:2.0/5 XIO I:2.0/4 NXB XIC I:2.0/4 XIC N7:76/6 NXB XIO I:1.0/0 NXB XIO I:1.0/1 NXB XIC I:2.0/10 BND OTU N7:51/6 EOR
%   I:2.0/5  BTN_REZIM_VYCH_POLOH %
%   I:2.0/4  BTN_REZIM_AUTOMAT %
%   I:1.0/0  BEZP_BRANKA_ZAVRENA %
%   I:1.0/1  HYDR_AGREGAT_CHOD %
%   I:2.0/10  BTN_STOP_AUTOMATU %
%   N7:51/6  REZIM_VYCHOZI_POLOHA %
% Rung: 76 %
SOR XIC I:2.0/7 XIC I:1.0/0 XIO I:2.0/8 XIO I:2.0/5 XIO I:2.0/4 OTE N7:51/5 EOR
%   I:2.0/7  BTN_REZIM_RUCNE %
%   I:1.0/0  BEZP_BRANKA_ZAVRENA %
%   I:2.0/8  INP_SERIZOVANI %
%   I:2.0/5  BTN_REZIM_VYCH_POLOH %
%   I:2.0/4  BTN_REZIM_AUTOMAT %
% Rung: 77 %
SOR XIC I:2.0/8 XIC I:2.0/3 XIO I:2.0/4 XIO I:2.0/7 XIO I:2.0/5 OTE N7:51/3 EOR
%   I:2.0/8  INP_SERIZOVANI %
%   I:2.0/3  INP_ZAMEK_SERIZOVANI %
%   I:2.0/4  BTN_REZIM_AUTOMAT %
%   I:2.0/7  BTN_REZIM_RUCNE %
%   I:2.0/5  BTN_REZIM_VYCH_POLOH %
%   N7:51/3  REZIM_SERIZOVANI %
% Rung: 78 %
SOR XIC N7:45/15 XIC N7:51/1 OTL N7:53/11 EOR
% Rung: 79 %
SOR BST XIC N7:45/15 XIC I:2.0/7 NXB XIC I:2.0/6 BND JSR U:14 EOR
%   I:2.0/7  BTN_REZIM_RUCNE %
% Rung: 80 %
SOR JSR U:5 EOR
% Rung: 81 %
SOR XIC N7:51/14 JSR U:6 EOR
% Rung: 82 %
SOR JSR U:7 EOR
% Rung: 83 %
SOR JSR U:8 EOR

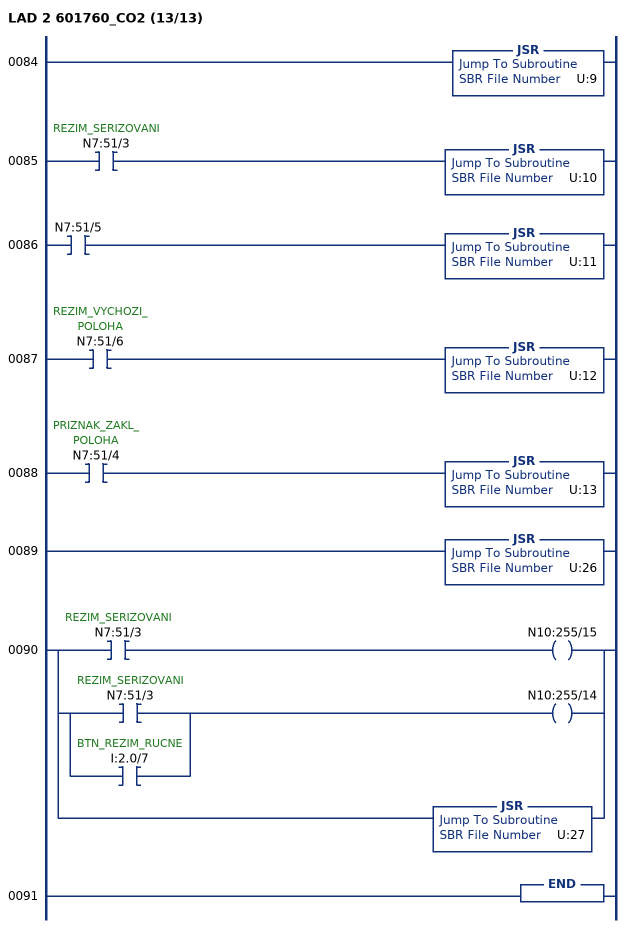
% Rung: 84 %
SOR JSR U:9 EOR
% Rung: 85 %
SOR XIC N7:51/3 JSR U:10 EOR
%   N7:51/3  REZIM_SERIZOVANI %
% Rung: 86 %
SOR XIC N7:51/5 JSR U:11 EOR
% Rung: 87 %
SOR XIC N7:51/6 JSR U:12 EOR
%   N7:51/6  REZIM_VYCHOZI_POLOHA %
% Rung: 88 %
SOR XIC N7:51/4 JSR U:13 EOR
%   N7:51/4  PRIZNAK_ZAKL_POLOHA %
% Rung: 89 %
SOR JSR U:26 EOR
% Rung: 90 %
SOR BST XIC N7:51/3 OTE N10:255/15 NXB BST XIC N7:51/3 NXB XIC I:2.0/7 BND OTE N10:255/14 NXB JSR U:27 BND EOR
%   N7:51/3  REZIM_SERIZOVANI %
%   I:2.0/7  BTN_REZIM_RUCNE %
% Rung: 91 %
SOR END EOR

LADDER 3
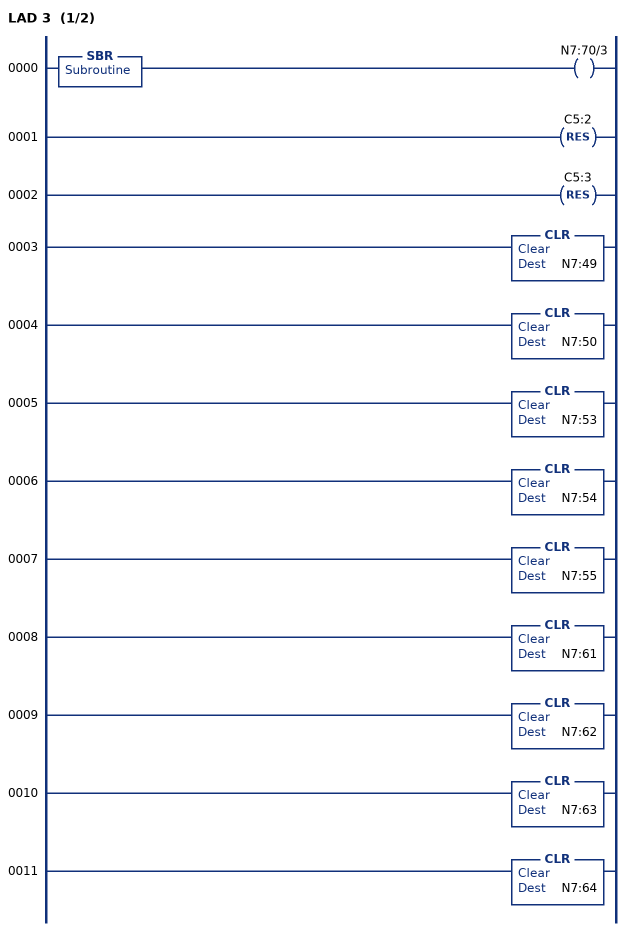
% Rung: 0 %
SOR SBR OTE N7:70/3 EOR
% Rung: 1 %
SOR RES C5:2 EOR
% Rung: 2 %
SOR RES C5:3 EOR
% Rung: 3 %
SOR CLR N7:49 EOR
% Rung: 4 %
SOR CLR N7:50 EOR
% Rung: 5 %
SOR CLR N7:53 EOR
% Rung: 6 %
SOR CLR N7:54 EOR
% Rung: 7 %
SOR CLR N7:55 EOR
% Rung: 8 %
SOR CLR N7:61 EOR
% Rung: 9 %
SOR CLR N7:62 EOR
% Rung: 10 %
SOR CLR N7:63 EOR
% Rung: 11 %
SOR CLR N7:64 EOR

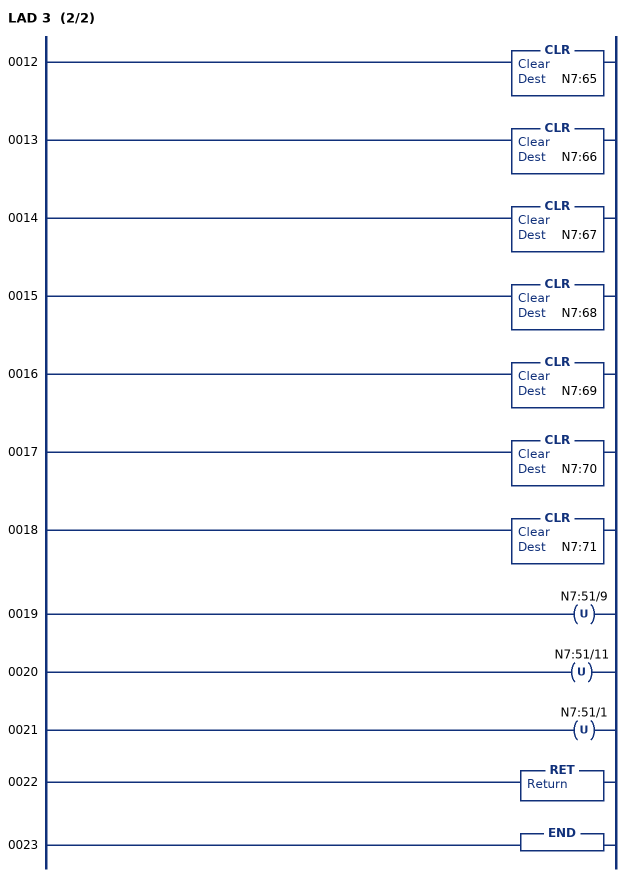
% Rung: 12 %
SOR CLR N7:65 EOR
% Rung: 13 %
SOR CLR N7:66 EOR
% Rung: 14 %
SOR CLR N7:67 EOR
% Rung: 15 %
SOR CLR N7:68 EOR
% Rung: 16 %
SOR CLR N7:69 EOR
% Rung: 17 %
SOR CLR N7:70 EOR
% Rung: 18 %
SOR CLR N7:71 EOR
% Rung: 19 %
SOR OTU N7:51/9 EOR
% Rung: 20 %
SOR OTU N7:51/11 EOR
% Rung: 21 %
SOR OTU N7:51/1 EOR
% Rung: 22 %
SOR RET EOR
% Rung: 23 %
SOR END EOR

LADDER 4
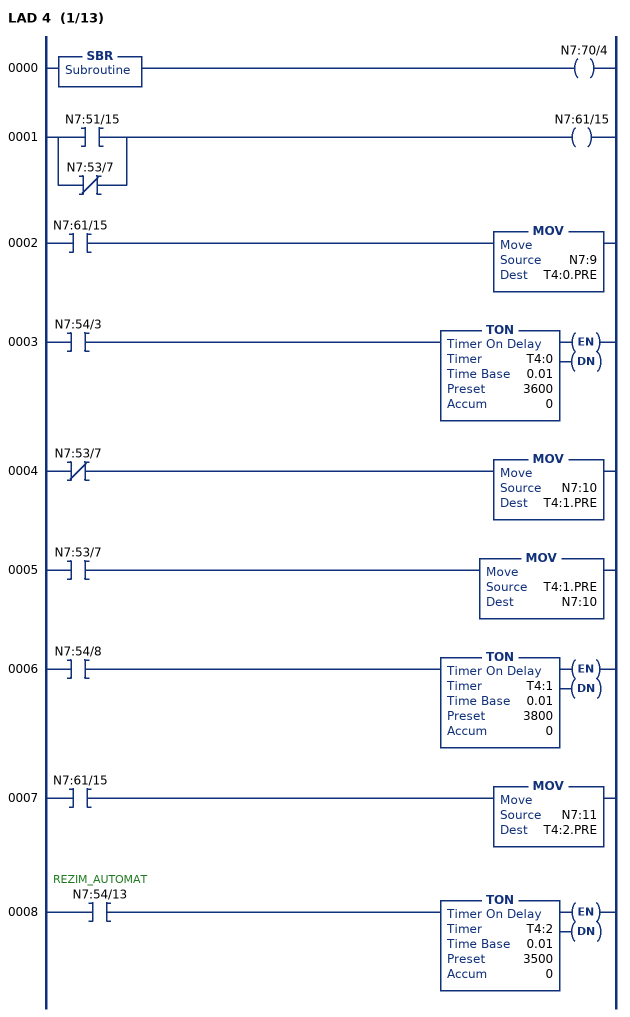
% Rung: 0 %
SOR SBR OTE N7:70/4 EOR
% Rung: 1 %
SOR BST XIC N7:51/15 NXB XIO N7:53/7 BND OTE N7:61/15 EOR
% Rung: 2 %
SOR XIC N7:61/15 MOV N7:9 T4:0.PRE EOR
% Rung: 3 %
SOR XIC N7:54/3 TON T4:0 0.01 3600 0 EOR
% Rung: 4 %
SOR XIO N7:53/7 MOV N7:10 T4:1.PRE EOR
% Rung: 5 %
SOR XIC N7:53/7 MOV T4:1.PRE N7:10 EOR
% Rung: 6 %
SOR XIC N7:54/8 TON T4:1 0.01 3800 0 EOR
% Rung: 7 %
SOR XIC N7:61/15 MOV N7:11 T4:2.PRE EOR
% Rung: 8 %
SOR XIC N7:54/13 TON T4:2 0.01 3500 0 EOR
%   N7:54/13  REZIM_AUTOMAT %

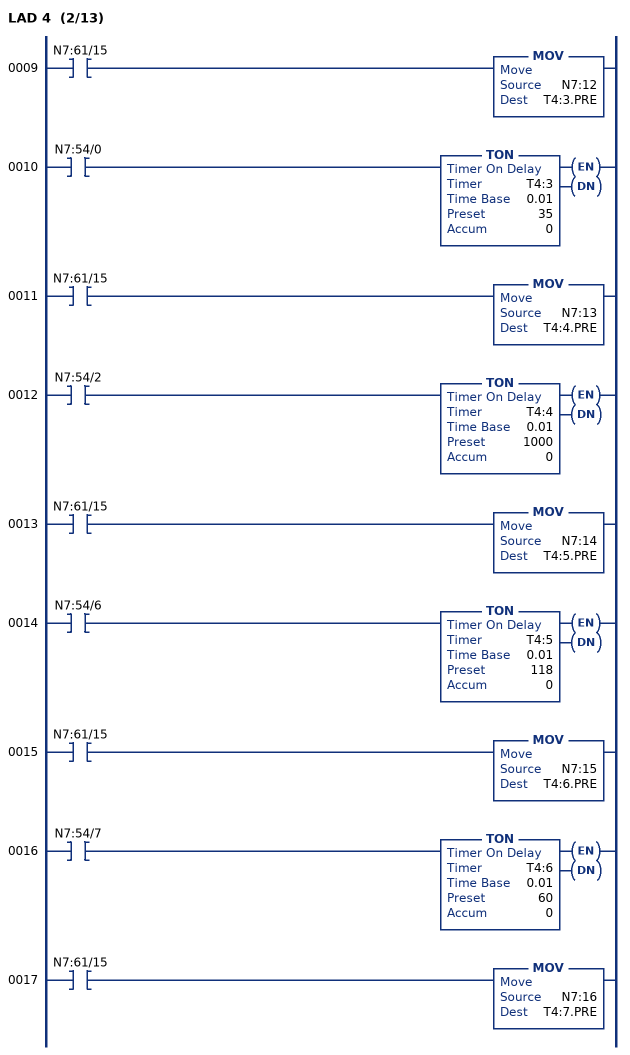
% Rung: 9 %
SOR XIC N7:61/15 MOV N7:12 T4:3.PRE EOR
% Rung: 10 %
SOR XIC N7:54/0 TON T4:3 0.01 35 0 EOR
% Rung: 11 %
SOR XIC N7:61/15 MOV N7:13 T4:4.PRE EOR
%   N7:13  TIM_KOPYTO_VPRED_PRE %
% Rung: 12 %
SOR XIC N7:54/2 TON T4:4 0.01 1000 0 EOR
% Rung: 13 %
SOR XIC N7:61/15 MOV N7:14 T4:5.PRE EOR
% Rung: 14 %
SOR XIC N7:54/6 TON T4:5 0.01 118 0 EOR
% Rung: 15 %
SOR XIC N7:61/15 MOV N7:15 T4:6.PRE EOR
% Rung: 16 %
SOR XIC N7:54/7 TON T4:6 0.01 60 0 EOR
% Rung: 17 %
SOR XIC N7:61/15 MOV N7:16 T4:7.PRE EOR

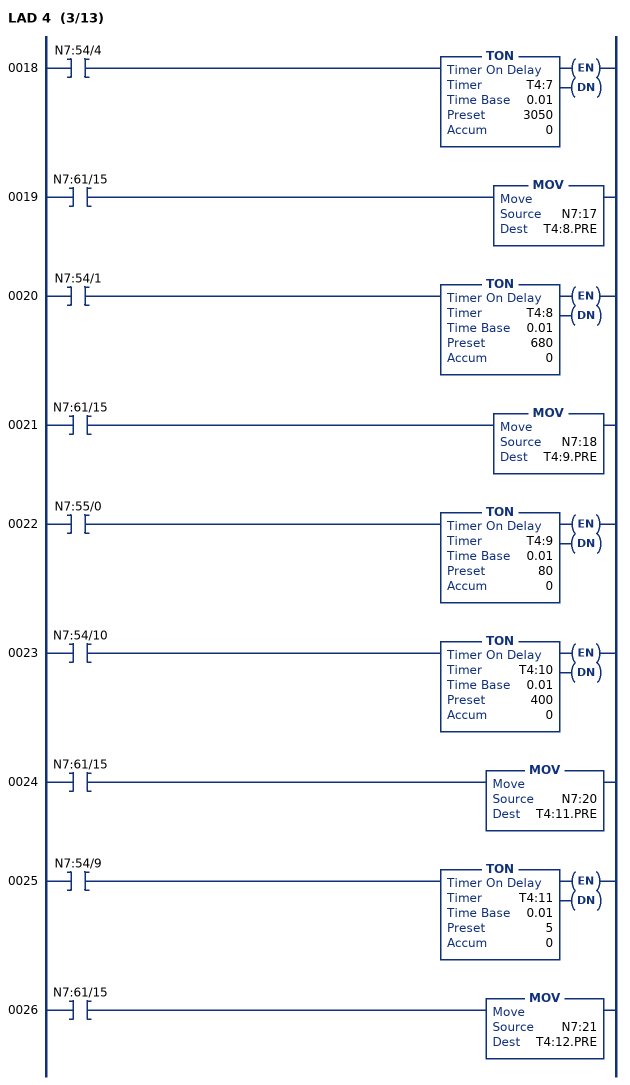
% Rung: 18 %
SOR XIC N7:54/4 TON T4:7 0.01 3050 0 EOR
% Rung: 19 %
SOR XIC N7:61/15 MOV N7:17 T4:8.PRE EOR
% Rung: 20 %
SOR XIC N7:54/1 TON T4:8 0.01 680 0 EOR
% Rung: 21 %
SOR XIC N7:61/15 MOV N7:18 T4:9.PRE EOR
% Rung: 22 %
SOR XIC N7:55/0 TON T4:9 0.01 80 0 EOR
% Rung: 23 %
SOR XIC N7:54/10 TON T4:10 0.01 400 0 EOR
% Rung: 24 %
SOR XIC N7:61/15 MOV N7:20 T4:11.PRE EOR
% Rung: 25 %
SOR XIC N7:54/9 TON T4:11 0.01 5 0 EOR
% Rung: 26 %
SOR XIC N7:61/15 MOV N7:21 T4:12.PRE EOR

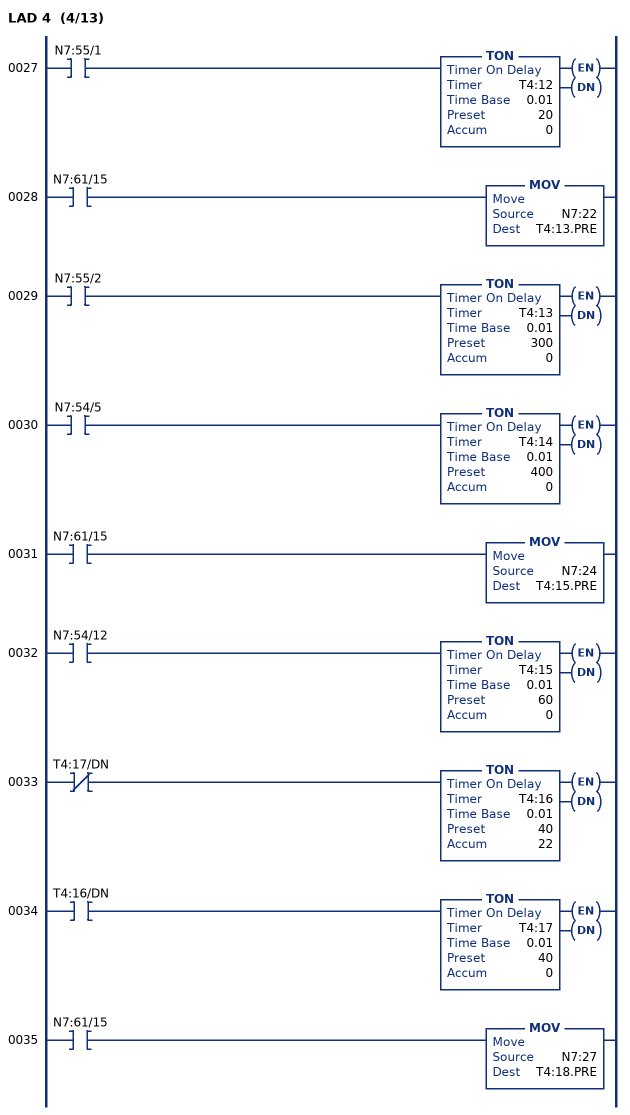
% Rung: 27 %
SOR XIC N7:55/1 TON T4:12 0.01 20 0 EOR
% Rung: 28 %
SOR XIC N7:61/15 MOV N7:22 T4:13.PRE EOR
% Rung: 29 %
SOR XIC N7:55/2 TON T4:13 0.01 300 0 EOR
% Rung: 30 %
SOR XIC N7:54/5 TON T4:14 0.01 400 0 EOR
% Rung: 31 %
SOR XIC N7:61/15 MOV N7:24 T4:15.PRE EOR
% Rung: 32 %
SOR XIC N7:54/12 TON T4:15 0.01 60 0 EOR
% Rung: 33 %
SOR XIO T4:17/DN TON T4:16 0.01 40 22 EOR
% Rung: 34 %
SOR XIC T4:16/DN TON T4:17 0.01 40 0 EOR
% Rung: 35 %
SOR XIC N7:61/15 MOV N7:27 T4:18.PRE EOR

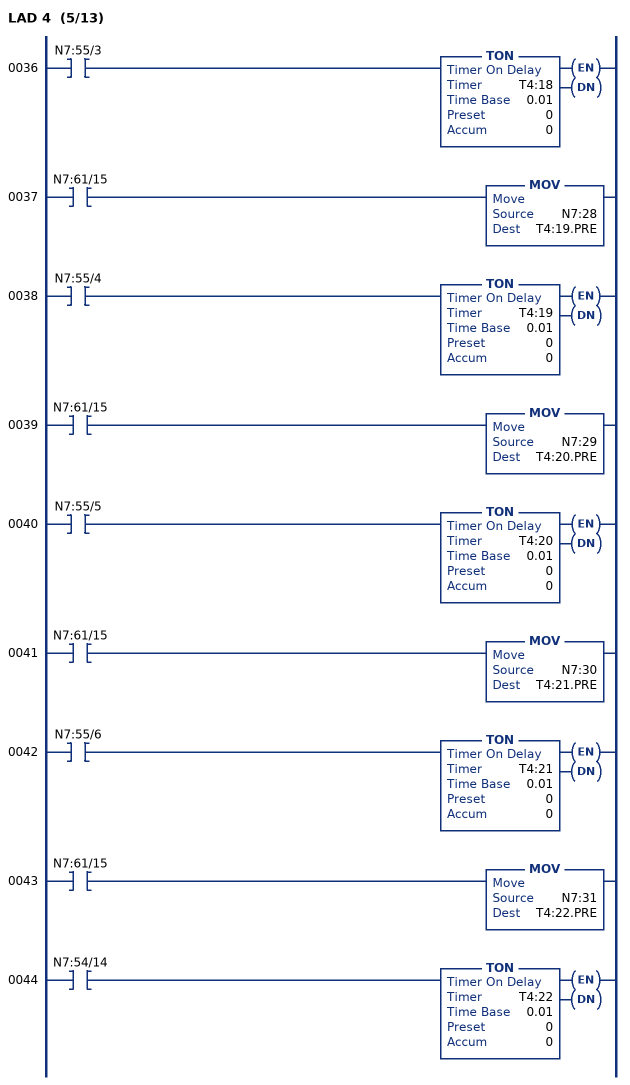
% Rung: 36 %
SOR XIC N7:55/3 TON T4:18 0.01 0 0 EOR
% Rung: 37 %
SOR XIC N7:61/15 MOV N7:28 T4:19.PRE EOR
% Rung: 38 %
SOR XIC N7:55/4 TON T4:19 0.01 0 0 EOR
% Rung: 39 %
SOR XIC N7:61/15 MOV N7:29 T4:20.PRE EOR
% Rung: 40 %
SOR XIC N7:55/5 TON T4:20 0.01 0 0 EOR
% Rung: 41 %
SOR XIC N7:61/15 MOV N7:30 T4:21.PRE EOR
% Rung: 42 %
SOR XIC N7:55/6 TON T4:21 0.01 0 0 EOR
% Rung: 43 %
SOR XIC N7:61/15 MOV N7:31 T4:22.PRE EOR
% Rung: 44 %
SOR XIC N7:54/14 TON T4:22 0.01 0 0 EOR

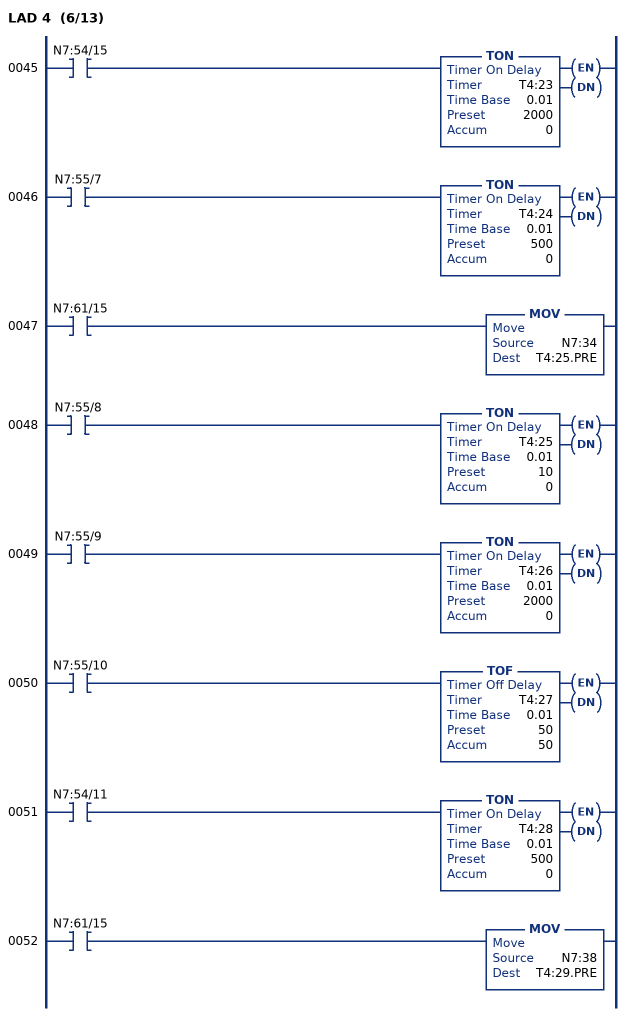
% Rung: 45 %
SOR XIC N7:54/15 TON T4:23 0.01 2000 0 EOR
% Rung: 46 %
SOR XIC N7:55/7 TON T4:24 0.01 500 0 EOR
% Rung: 47 %
SOR XIC N7:61/15 MOV N7:34 T4:25.PRE EOR
% Rung: 48 %
SOR XIC N7:55/8 TON T4:25 0.01 10 0 EOR
% Rung: 49 %
SOR XIC N7:55/9 TON T4:26 0.01 2000 0 EOR
% Rung: 50 %
SOR XIC N7:55/10 TOF T4:27 0.01 50 50 EOR
% Rung: 51 %
SOR XIC N7:54/11 TON T4:28 0.01 500 0 EOR
% Rung: 52 %
SOR XIC N7:61/15 MOV N7:38 T4:29.PRE EOR

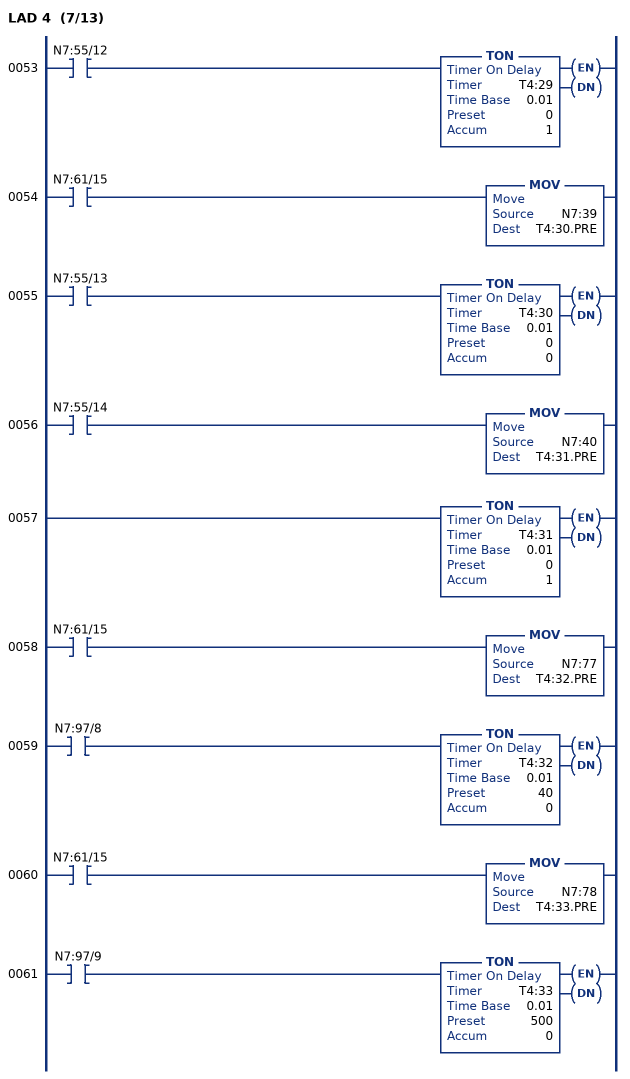
% Rung: 53 %
SOR XIC N7:55/12 TON T4:29 0.01 0 1 EOR
% Rung: 54 %
SOR XIC N7:61/15 MOV N7:39 T4:30.PRE EOR
% Rung: 55 %
SOR XIC N7:55/13 TON T4:30 0.01 0 0 EOR
% Rung: 56 %
SOR XIC N7:55/14 MOV N7:40 T4:31.PRE EOR
% Rung: 57 %
SOR TON T4:31 0.01 0 1 EOR
% Rung: 58 %
SOR XIC N7:61/15 MOV N7:77 T4:32.PRE EOR
% Rung: 59 %
SOR XIC N7:97/8 TON T4:32 0.01 40 0 EOR
% Rung: 60 %
SOR XIC N7:61/15 MOV N7:78 T4:33.PRE EOR
% Rung: 61 %
SOR XIC N7:97/9 TON T4:33 0.01 500 0 EOR

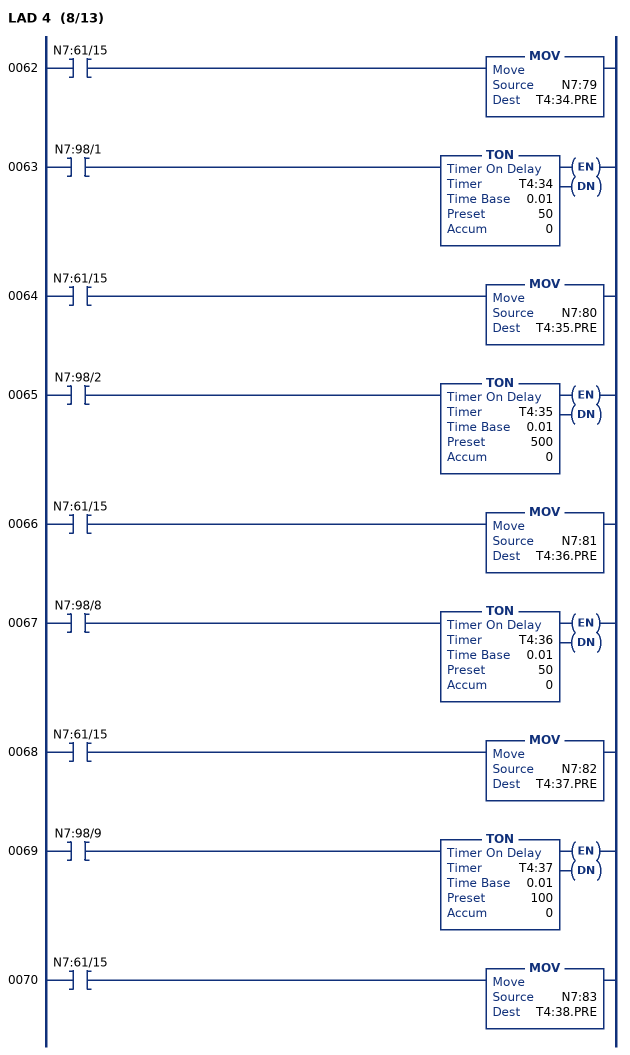
% Rung: 62 %
SOR XIC N7:61/15 MOV N7:79 T4:34.PRE EOR
% Rung: 63 %
SOR XIC N7:98/1 TON T4:34 0.01 50 0 EOR
% Rung: 64 %
SOR XIC N7:61/15 MOV N7:80 T4:35.PRE EOR
% Rung: 65 %
SOR XIC N7:98/2 TON T4:35 0.01 500 0 EOR
% Rung: 66 %
SOR XIC N7:61/15 MOV N7:81 T4:36.PRE EOR
% Rung: 67 %
SOR XIC N7:98/8 TON T4:36 0.01 50 0 EOR
% Rung: 68 %
SOR XIC N7:61/15 MOV N7:82 T4:37.PRE EOR
% Rung: 69 %
SOR XIC N7:98/9 TON T4:37 0.01 100 0 EOR
% Rung: 70 %
SOR XIC N7:61/15 MOV N7:83 T4:38.PRE EOR

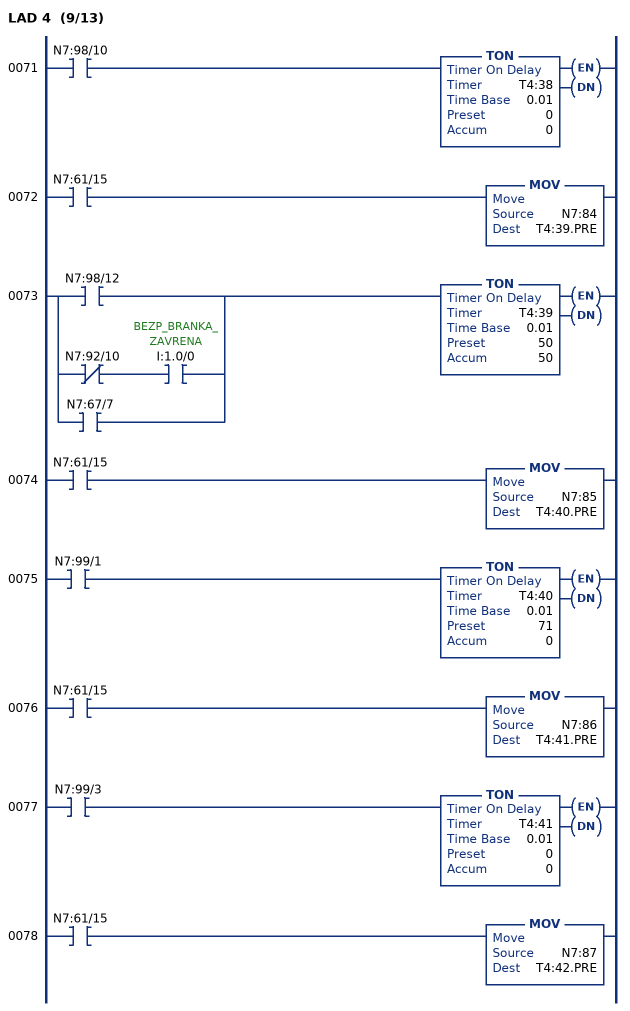
% Rung: 71 %
SOR XIC N7:98/10 TON T4:38 0.01 0 0 EOR
% Rung: 72 %
SOR XIC N7:61/15 MOV N7:84 T4:39.PRE EOR
% Rung: 73 %
SOR BST XIC N7:98/12 NXB XIO N7:92/10 XIC I:1.0/0 NXB XIC N7:67/7 BND TON T4:39 0.01 50 50 EOR
%   I:1.0/0  BEZP_BRANKA_ZAVRENA %
% Rung: 74 %
SOR XIC N7:61/15 MOV N7:85 T4:40.PRE EOR
% Rung: 75 %
SOR XIC N7:99/1 TON T4:40 0.01 71 0 EOR
% Rung: 76 %
SOR XIC N7:61/15 MOV N7:86 T4:41.PRE EOR
% Rung: 77 %
SOR XIC N7:99/3 TON T4:41 0.01 0 0 EOR
% Rung: 78 %
SOR XIC N7:61/15 MOV N7:87 T4:42.PRE EOR

